{attribute addProperty BoxType "EK1122-0000-0018"}
{attribute addProperty Id "Beckhoff_EL47xxsub_EK1100EK1100_179A0949162"}
{attribute addProperty CRC "1257898769"}
{attribute addProperty SizeInBites "16"}
{attribute addProperty SizeInBytes "2"}
TYPE Beckhoff_EL47xxEK1122_4AFA0311 EXTENDS EK1122_179A0949 :
STRUCT
	{attribute addProperty Name "Beckhoff_EL47xxsub_EK1100"}
	Beckhoff_EL47xxsub_EK1100 : EK1100_179A0949;
END_STRUCT
END_TYPE

(* stored: Version 1.2.0.0, ProductVersion 3.1.4024.9
   DUT Beckhoff_EL47xxEK1122_4AFA0311: Id {7c10e7af-1d72-4192-a30b-1f9faecc35aa} *)
